// TIA Portal V19 export
DATA_BLOCK "PUT_Request_DB"   // DB9
// stored: InstanceOfName PUT_Request, InstanceOfType FB
"PUT_Request"
   // VAR_INPUT
   //    start : Bool;
   //    url : String;
   //    data : String;
   // END_VAR
   // VAR_OUTPUT
   //    connected : Bool;
   //    done : Bool;
   //    busy : Bool;
   //    error : Bool;
   //    status : Word;
   //    diagnostics : "typeDiagnostics";
   //    responseCode : UInt;
   //    length : UDInt;
   // END_VAR
   // VAR_IN_OUT
   //    responseData : Array[0..255] of Char;
   // END_VAR
   // VAR
   //    hwID : HW_ANY;
   //    connID : CONN_OUC := 16#0002;
   //    keepConnection : Bool;
   // END_VAR
BEGIN
END_DATA_BLOCK
